(* Logix 5000 project; controller cal1615 1756-L62 rev 16.20; software revision 16.05; part 47 of 78 *)
(* tags used below, declared in another part *)
   FAULT : BOOL;   // Fault AFI
   HMI : BOOL;   // AFI HMI
   p01r03_lc3_ave_ctrl : CONTROL;
   p01r09_pb_global_reset : BOOL;   // System Modes PB: Global Fault Reset
   p02_real_from_hmi : hmi_real;   // MOP HMI Iface Real from HMI
   p22_ai_amps : REAL;   // Tension Stand 1 Analog Input Tension Stand 1 Motor Current
   p22_ai_hz : REAL;   // Tension Stand 1 Analog Input Tension Stand 1 Motor Hertz
   p22_ai_speed : REAL;
   p22_ai_ts1_lc : REAL;   // Tension Stand 1 Analog Input Loadcell
   p22_ao_selected_speed : REAL;   // Tension Stand 1 VFD Selected Speed
   p22_dint_to_hmi : DINT[16];   // Tension Stand 1 Dint to HMI
   p22_real_to_hmi : REAL[112];   // Tension Stand 1 Real to HMI
   p22r01 : routine;   // Tension Stand 1 Main
   p22r06 : routine;   // Tension Stand 1 Real to HMI
   p22r06_ave_lc : REAL;
   p22r06_lc_buffer : REAL[20];
   p22r06_lc_ctrl : CONTROL;
   p22r06_sample_timer : TIMER;
   p22r06_timer_fault : TIMER[4];   // Tension Stand 1 Real to HMI Fault Delay
   p22r06_timer_warning : TIMER[4];   // Tension Stand 1 Real to HMI Warning Delay
   p22r06_unload : DINT;
   p22r07 : routine;   // Tension Stand 1 Alarms
   p22r07_timer_fault : TIMER[4];   // Tension Stand 1 Alarms Fault Delay
   p22r07_timer_warning : TIMER[4];   // Tension Stand 1 Alarms Warning Delay
   p22r08 : routine;   // Tension Stand 1 Warnings
   p22r08_timer_fault : TIMER[4];   // Tension Stand 1 Warnings Fault Delay
   p22r08_timer_warning : TIMER[4];   // Tension Stand 1 Warnings Warning Delay
   p22r09 : routine;   // Tension Stand 1 Modes
   p22r11 : routine;   // Tension Stand 1 VFD
(* P22_Tension_Stand_1, continued *)

ROUTINE R06_Real_to_HMI   (* ladder *)
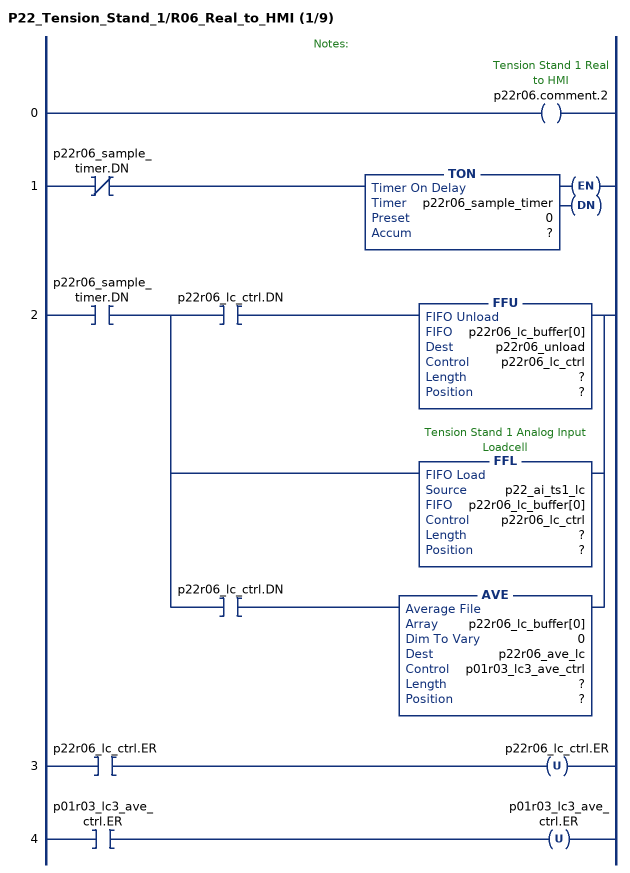
   // Notes:
   0: OTE(p22r06.comment.2);
   1: XIO(p22r06_sample_timer.DN)TON(p22r06_sample_timer,?,?);
   2: XIC(p22r06_sample_timer.DN)[XIC(p22r06_lc_ctrl.DN) FFU(p22r06_lc_buffer[0],p22r06_unload,p22r06_lc_ctrl,?,?) ,FFL(p22_ai_ts1_lc,p22r06_lc_buffer[0],p22r06_lc_ctrl,?,?) ,XIC(p22r06_lc_ctrl.DN) AVE(p22r06_lc_buffer[0],0,p22r06_ave_lc,p01r03_lc3_ave_ctrl,?,?) ];
   3: XIC(p22r06_lc_ctrl.ER)OTU(p22r06_lc_ctrl.ER);
   4: XIC(p01r03_lc3_ave_ctrl.ER)OTU(p01r03_lc3_ave_ctrl.ER);
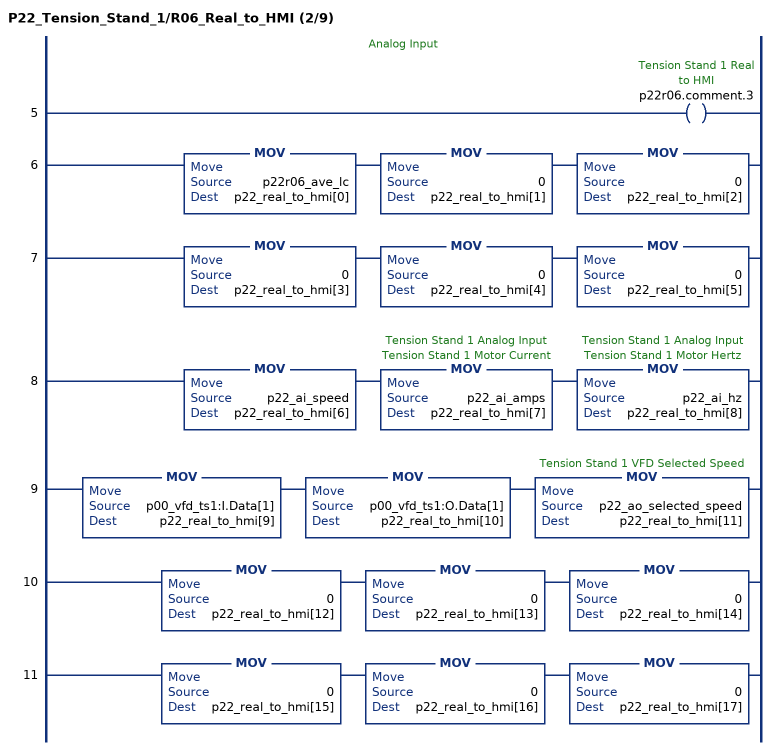
   // Analog Input
   5: OTE(p22r06.comment.3);
   6: MOV(p22r06_ave_lc,p22_real_to_hmi[0])MOV(0,p22_real_to_hmi[1])MOV(0,p22_real_to_hmi[2]);
   7: MOV(0,p22_real_to_hmi[3])MOV(0,p22_real_to_hmi[4])MOV(0,p22_real_to_hmi[5]);
   8: MOV(p22_ai_speed,p22_real_to_hmi[6])MOV(p22_ai_amps,p22_real_to_hmi[7])MOV(p22_ai_hz,p22_real_to_hmi[8]);
   9: MOV(p00_vfd_ts1:I.Data[1],p22_real_to_hmi[9])MOV(p00_vfd_ts1:O.Data[1],p22_real_to_hmi[10])MOV(p22_ao_selected_speed,p22_real_to_hmi[11]);
   10: MOV(0,p22_real_to_hmi[12])MOV(0,p22_real_to_hmi[13])MOV(0,p22_real_to_hmi[14]);
   11: MOV(0,p22_real_to_hmi[15])MOV(0,p22_real_to_hmi[16])MOV(0,p22_real_to_hmi[17]);
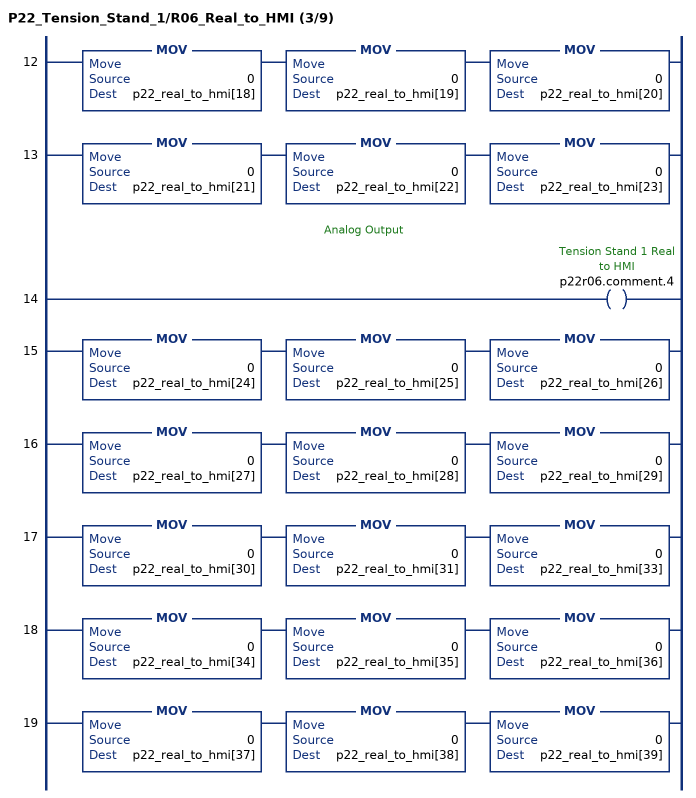
   12: MOV(0,p22_real_to_hmi[18])MOV(0,p22_real_to_hmi[19])MOV(0,p22_real_to_hmi[20]);
   13: MOV(0,p22_real_to_hmi[21])MOV(0,p22_real_to_hmi[22])MOV(0,p22_real_to_hmi[23]);
   // Analog Output
   14: OTE(p22r06.comment.4);
   15: MOV(0,p22_real_to_hmi[24])MOV(0,p22_real_to_hmi[25])MOV(0,p22_real_to_hmi[26]);
   16: MOV(0,p22_real_to_hmi[27])MOV(0,p22_real_to_hmi[28])MOV(0,p22_real_to_hmi[29]);
   17: MOV(0,p22_real_to_hmi[30])MOV(0,p22_real_to_hmi[31])MOV(0,p22_real_to_hmi[33]);
   18: MOV(0,p22_real_to_hmi[34])MOV(0,p22_real_to_hmi[35])MOV(0,p22_real_to_hmi[36]);
   19: MOV(0,p22_real_to_hmi[37])MOV(0,p22_real_to_hmi[38])MOV(0,p22_real_to_hmi[39]);
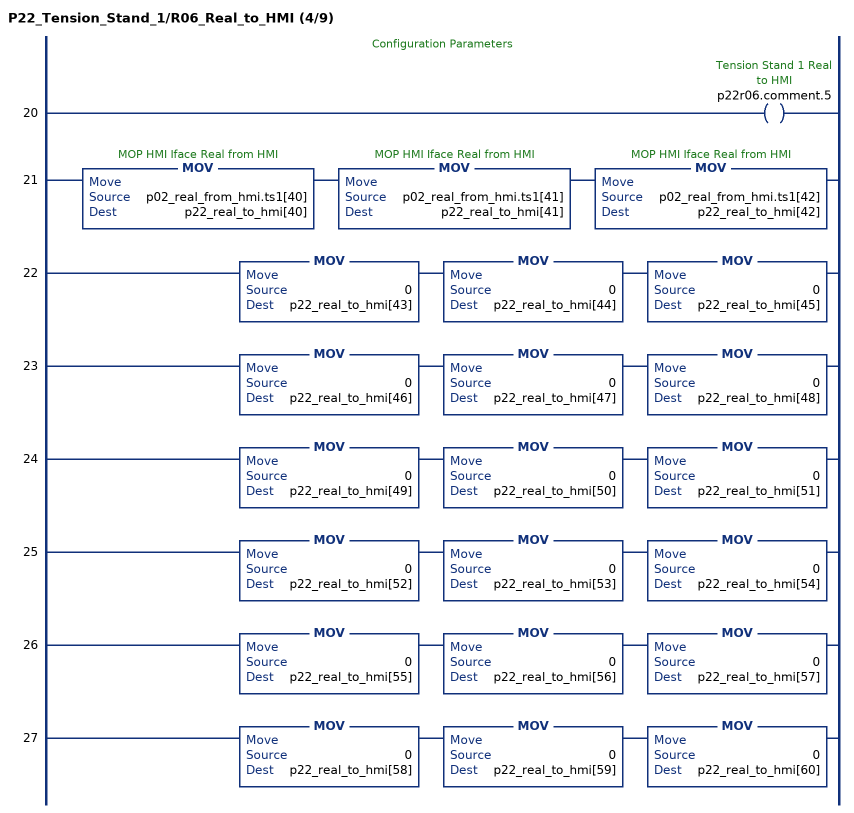
   // Configuration Parameters
   20: OTE(p22r06.comment.5);
   21: MOV(p02_real_from_hmi.ts1[40],p22_real_to_hmi[40])MOV(p02_real_from_hmi.ts1[41],p22_real_to_hmi[41])MOV(p02_real_from_hmi.ts1[42],p22_real_to_hmi[42]);
   22: MOV(0,p22_real_to_hmi[43])MOV(0,p22_real_to_hmi[44])MOV(0,p22_real_to_hmi[45]);
   23: MOV(0,p22_real_to_hmi[46])MOV(0,p22_real_to_hmi[47])MOV(0,p22_real_to_hmi[48]);
   24: MOV(0,p22_real_to_hmi[49])MOV(0,p22_real_to_hmi[50])MOV(0,p22_real_to_hmi[51]);
   25: MOV(0,p22_real_to_hmi[52])MOV(0,p22_real_to_hmi[53])MOV(0,p22_real_to_hmi[54]);
   26: MOV(0,p22_real_to_hmi[55])MOV(0,p22_real_to_hmi[56])MOV(0,p22_real_to_hmi[57]);
   27: MOV(0,p22_real_to_hmi[58])MOV(0,p22_real_to_hmi[59])MOV(0,p22_real_to_hmi[60]);
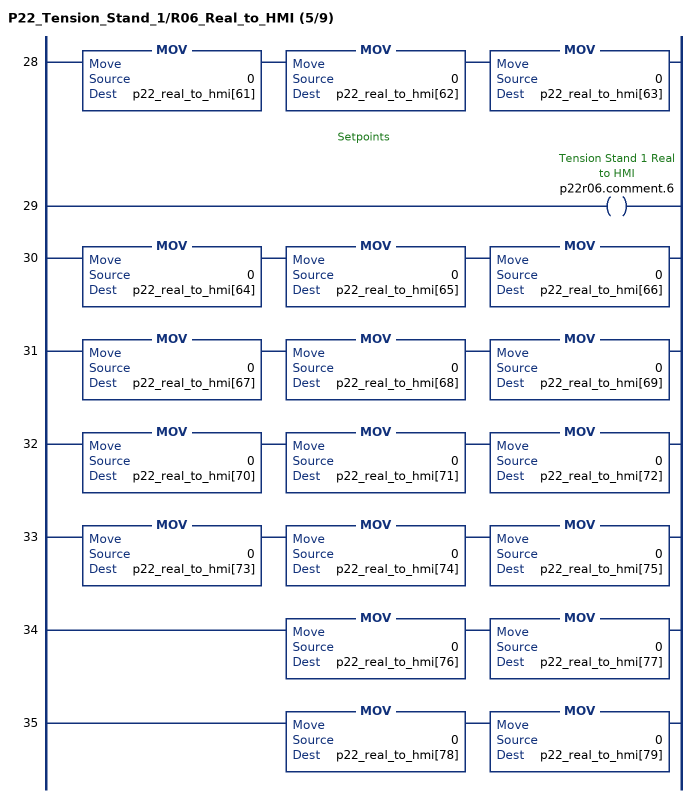
   28: MOV(0,p22_real_to_hmi[61])MOV(0,p22_real_to_hmi[62])MOV(0,p22_real_to_hmi[63]);
   // Setpoints
   29: OTE(p22r06.comment.6);
   30: MOV(0,p22_real_to_hmi[64])MOV(0,p22_real_to_hmi[65])MOV(0,p22_real_to_hmi[66]);
   31: MOV(0,p22_real_to_hmi[67])MOV(0,p22_real_to_hmi[68])MOV(0,p22_real_to_hmi[69]);
   32: MOV(0,p22_real_to_hmi[70])MOV(0,p22_real_to_hmi[71])MOV(0,p22_real_to_hmi[72]);
   33: MOV(0,p22_real_to_hmi[73])MOV(0,p22_real_to_hmi[74])MOV(0,p22_real_to_hmi[75]);
   34: MOV(0,p22_real_to_hmi[76])MOV(0,p22_real_to_hmi[77]);
   35: MOV(0,p22_real_to_hmi[78])MOV(0,p22_real_to_hmi[79]);
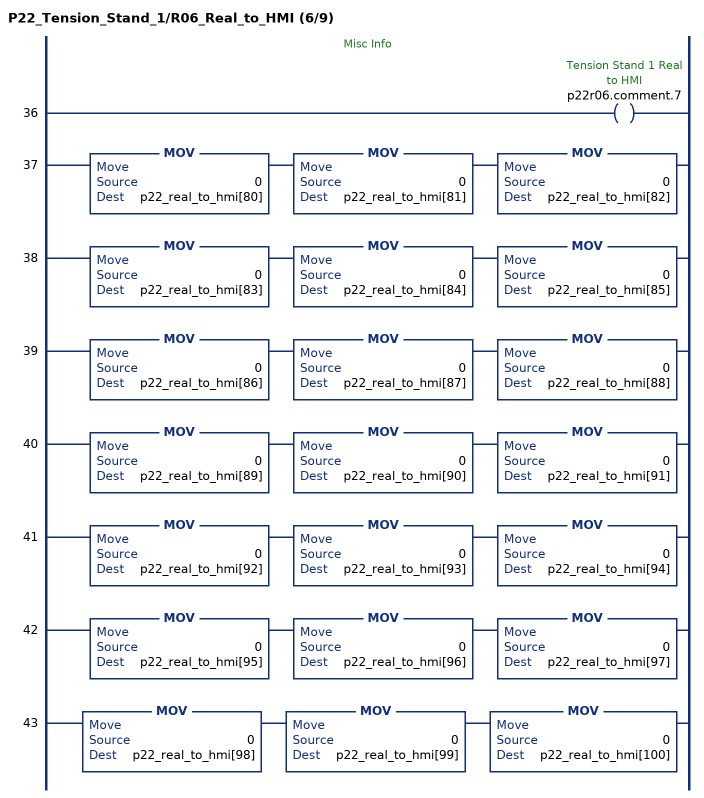
   // Misc Info
   36: OTE(p22r06.comment.7);
   37: MOV(0,p22_real_to_hmi[80])MOV(0,p22_real_to_hmi[81])MOV(0,p22_real_to_hmi[82]);
   38: MOV(0,p22_real_to_hmi[83])MOV(0,p22_real_to_hmi[84])MOV(0,p22_real_to_hmi[85]);
   39: MOV(0,p22_real_to_hmi[86])MOV(0,p22_real_to_hmi[87])MOV(0,p22_real_to_hmi[88]);
   40: MOV(0,p22_real_to_hmi[89])MOV(0,p22_real_to_hmi[90])MOV(0,p22_real_to_hmi[91]);
   41: MOV(0,p22_real_to_hmi[92])MOV(0,p22_real_to_hmi[93])MOV(0,p22_real_to_hmi[94]);
   42: MOV(0,p22_real_to_hmi[95])MOV(0,p22_real_to_hmi[96])MOV(0,p22_real_to_hmi[97]);
   43: MOV(0,p22_real_to_hmi[98])MOV(0,p22_real_to_hmi[99])MOV(0,p22_real_to_hmi[100]);
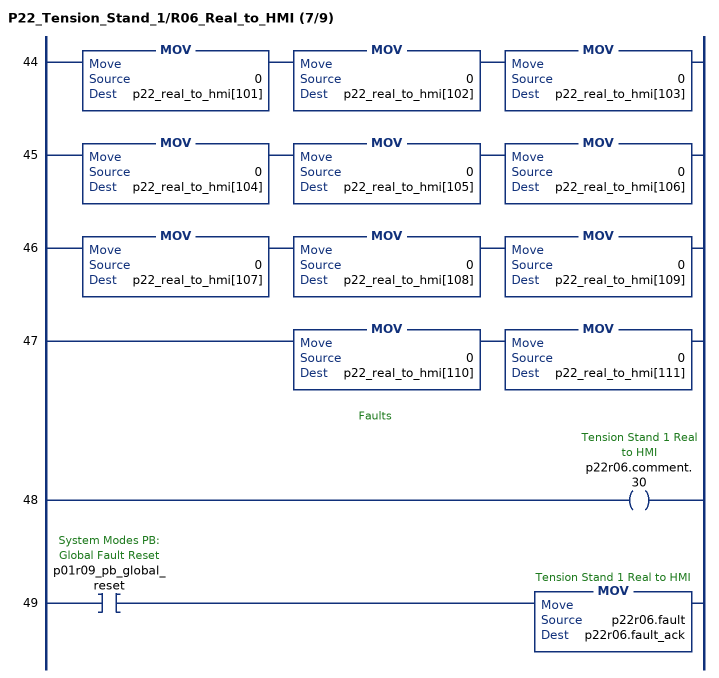
   44: MOV(0,p22_real_to_hmi[101])MOV(0,p22_real_to_hmi[102])MOV(0,p22_real_to_hmi[103]);
   45: MOV(0,p22_real_to_hmi[104])MOV(0,p22_real_to_hmi[105])MOV(0,p22_real_to_hmi[106]);
   46: MOV(0,p22_real_to_hmi[107])MOV(0,p22_real_to_hmi[108])MOV(0,p22_real_to_hmi[109]);
   47: MOV(0,p22_real_to_hmi[110])MOV(0,p22_real_to_hmi[111]);
   // Faults
   48: OTE(p22r06.comment.30);
   49: XIC(p01r09_pb_global_reset)MOV(p22r06.fault,p22r06.fault_ack);
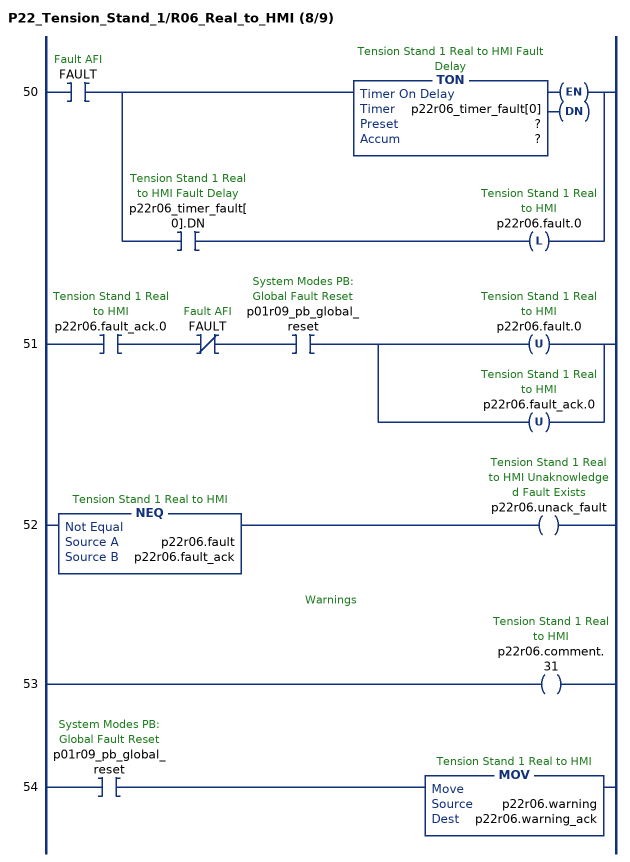
   50: XIC(FAULT)[TON(p22r06_timer_fault[0],?,?) ,XIC(p22r06_timer_fault[0].DN) OTL(p22r06.fault.0) ];
   51: XIC(p22r06.fault_ack.0)XIO(FAULT)XIC(p01r09_pb_global_reset)[OTU(p22r06.fault.0) ,OTU(p22r06.fault_ack.0) ];
   52: NEQ(p22r06.fault,p22r06.fault_ack)OTE(p22r06.unack_fault);
   // Warnings
   53: OTE(p22r06.comment.31);
   54: XIC(p01r09_pb_global_reset)MOV(p22r06.warning,p22r06.warning_ack);
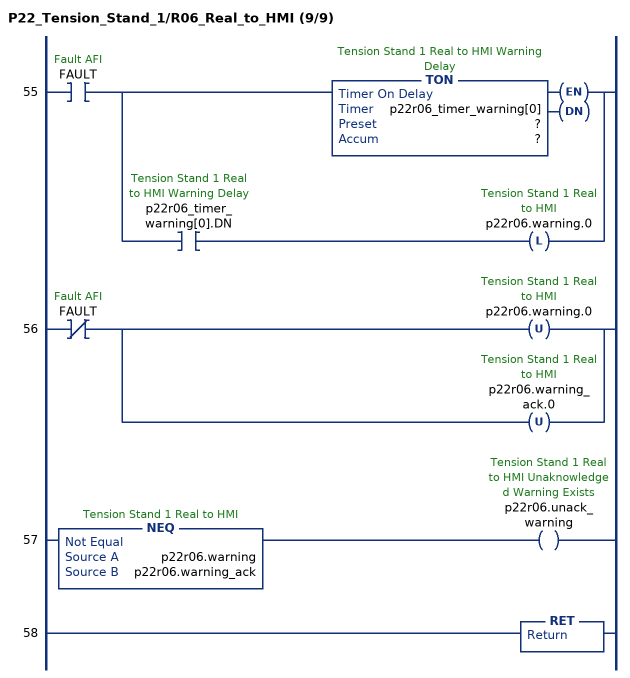
   55: XIC(FAULT)[TON(p22r06_timer_warning[0],?,?) ,XIC(p22r06_timer_warning[0].DN) OTL(p22r06.warning.0) ];
   56: XIO(FAULT)[OTU(p22r06.warning.0) ,OTU(p22r06.warning_ack.0) ];
   57: NEQ(p22r06.warning,p22r06.warning_ack)OTE(p22r06.unack_warning);
   58: RET();
END_ROUTINE

ROUTINE R07_Alarms   (* ladder *)
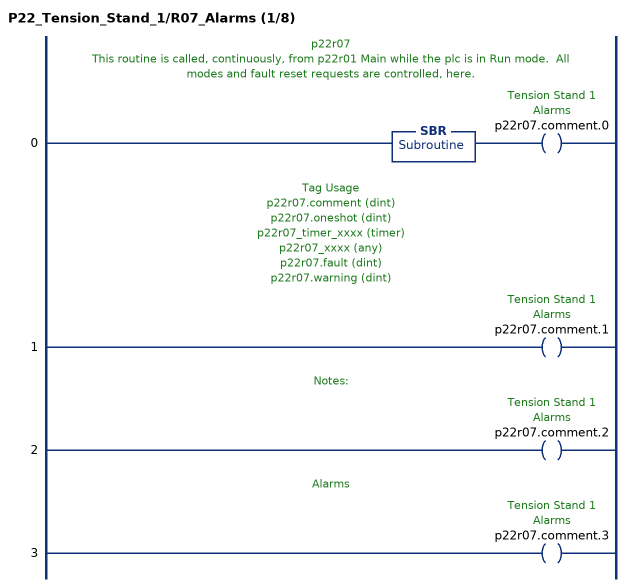
   // p22r07
   // This routine is called, continuously, from p22r01 Main while the plc is in Run mode.  All modes and fault reset requests are controlled, here.
   0: SBR()OTE(p22r07.comment.0);
   // Tag Usage
   // p22r07.comment (dint)
   // p22r07.oneshot (dint)
   // p22r07_timer_xxxx (timer)
   // p22r07_xxxx (any)
   // p22r07.fault (dint)
   // p22r07.warning (dint)
   1: OTE(p22r07.comment.1);
   // Notes:
   2: OTE(p22r07.comment.2);
   // Alarms
   3: OTE(p22r07.comment.3);
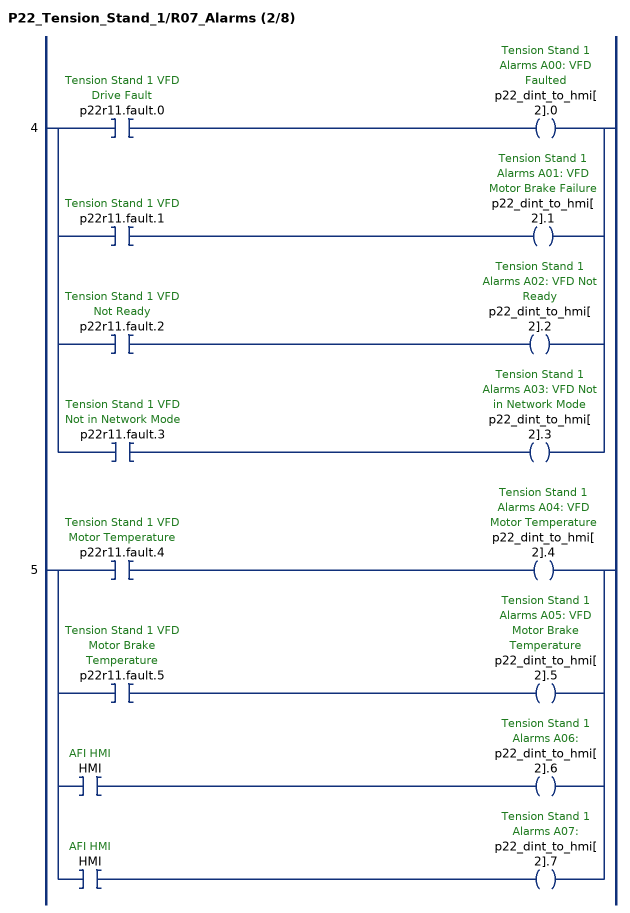
   4: [XIC(p22r11.fault.0) OTE(p22_dint_to_hmi[2].0) ,XIC(p22r11.fault.1) OTE(p22_dint_to_hmi[2].1) ,XIC(p22r11.fault.2) OTE(p22_dint_to_hmi[2].2) ,XIC(p22r11.fault.3) OTE(p22_dint_to_hmi[2].3) ];
   5: [XIC(p22r11.fault.4) OTE(p22_dint_to_hmi[2].4) ,XIC(p22r11.fault.5) OTE(p22_dint_to_hmi[2].5) ,XIC(HMI) OTE(p22_dint_to_hmi[2].6) ,XIC(HMI) OTE(p22_dint_to_hmi[2].7) ];
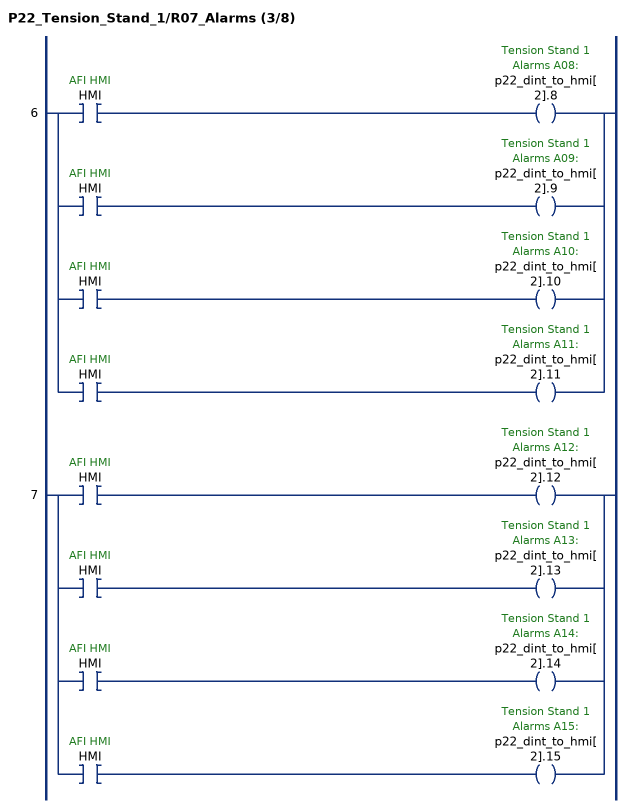
   6: [XIC(HMI) OTE(p22_dint_to_hmi[2].8) ,XIC(HMI) OTE(p22_dint_to_hmi[2].9) ,XIC(HMI) OTE(p22_dint_to_hmi[2].10) ,XIC(HMI) OTE(p22_dint_to_hmi[2].11) ];
   7: [XIC(HMI) OTE(p22_dint_to_hmi[2].12) ,XIC(HMI) OTE(p22_dint_to_hmi[2].13) ,XIC(HMI) OTE(p22_dint_to_hmi[2].14) ,XIC(HMI) OTE(p22_dint_to_hmi[2].15) ];
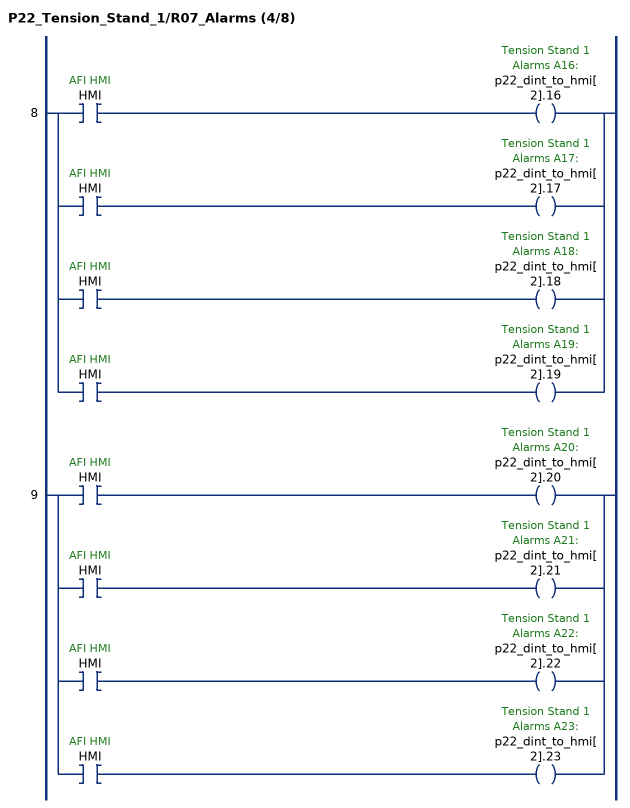
   8: [XIC(HMI) OTE(p22_dint_to_hmi[2].16) ,XIC(HMI) OTE(p22_dint_to_hmi[2].17) ,XIC(HMI) OTE(p22_dint_to_hmi[2].18) ,XIC(HMI) OTE(p22_dint_to_hmi[2].19) ];
   9: [XIC(HMI) OTE(p22_dint_to_hmi[2].20) ,XIC(HMI) OTE(p22_dint_to_hmi[2].21) ,XIC(HMI) OTE(p22_dint_to_hmi[2].22) ,XIC(HMI) OTE(p22_dint_to_hmi[2].23) ];
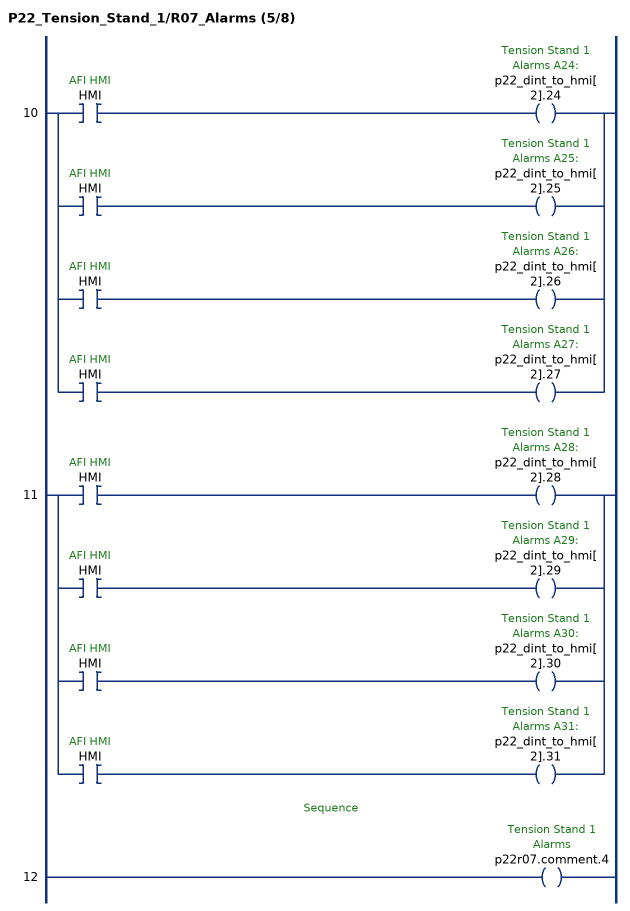
   10: [XIC(HMI) OTE(p22_dint_to_hmi[2].24) ,XIC(HMI) OTE(p22_dint_to_hmi[2].25) ,XIC(HMI) OTE(p22_dint_to_hmi[2].26) ,XIC(HMI) OTE(p22_dint_to_hmi[2].27) ];
   11: [XIC(HMI) OTE(p22_dint_to_hmi[2].28) ,XIC(HMI) OTE(p22_dint_to_hmi[2].29) ,XIC(HMI) OTE(p22_dint_to_hmi[2].30) ,XIC(HMI) OTE(p22_dint_to_hmi[2].31) ];
   // Sequence
   12: OTE(p22r07.comment.4);
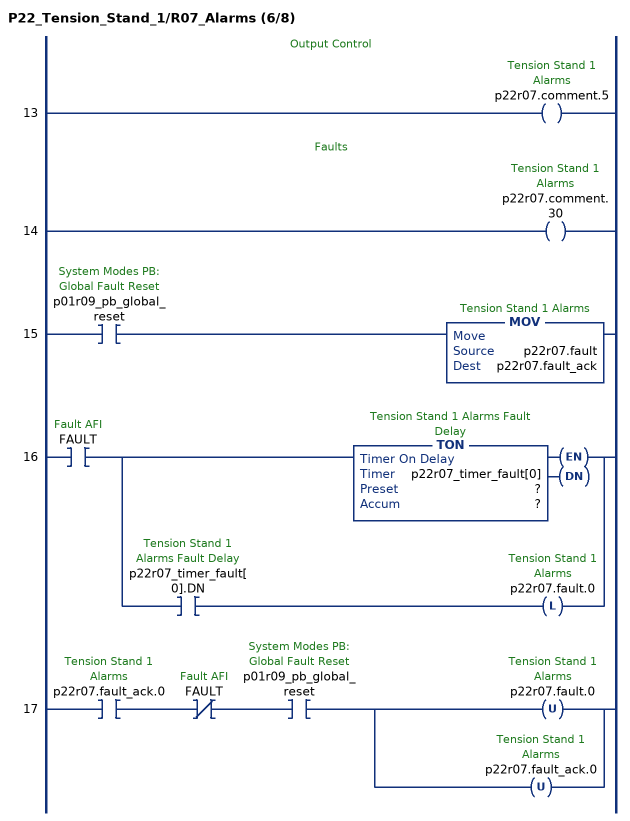
   // Output Control
   13: OTE(p22r07.comment.5);
   // Faults
   14: OTE(p22r07.comment.30);
   15: XIC(p01r09_pb_global_reset)MOV(p22r07.fault,p22r07.fault_ack);
   16: XIC(FAULT)[TON(p22r07_timer_fault[0],?,?) ,XIC(p22r07_timer_fault[0].DN) OTL(p22r07.fault.0) ];
   17: XIC(p22r07.fault_ack.0)XIO(FAULT)XIC(p01r09_pb_global_reset)[OTU(p22r07.fault.0) ,OTU(p22r07.fault_ack.0) ];
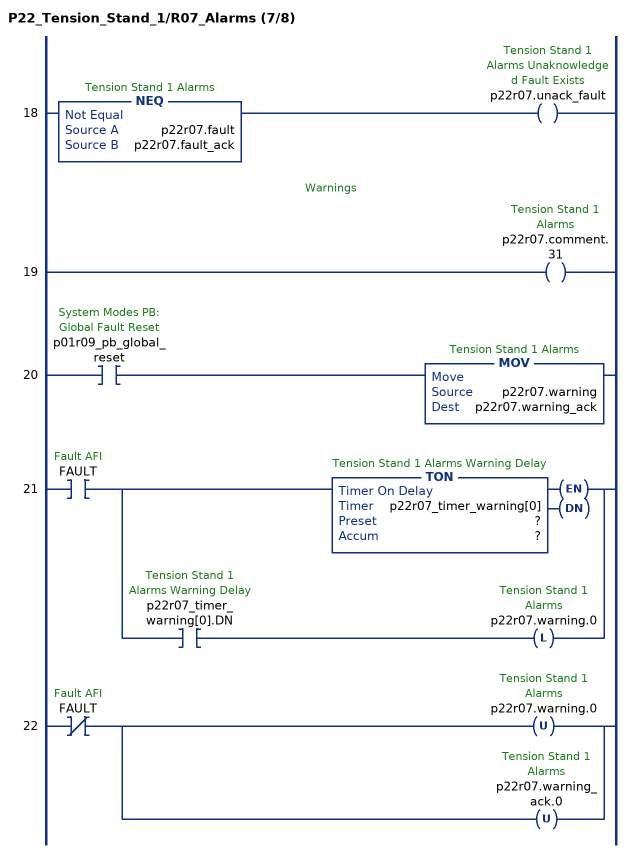
   18: NEQ(p22r07.fault,p22r07.fault_ack)OTE(p22r07.unack_fault);
   // Warnings
   19: OTE(p22r07.comment.31);
   20: XIC(p01r09_pb_global_reset)MOV(p22r07.warning,p22r07.warning_ack);
   21: XIC(FAULT)[TON(p22r07_timer_warning[0],?,?) ,XIC(p22r07_timer_warning[0].DN) OTL(p22r07.warning.0) ];
   22: XIO(FAULT)[OTU(p22r07.warning.0) ,OTU(p22r07.warning_ack.0) ];
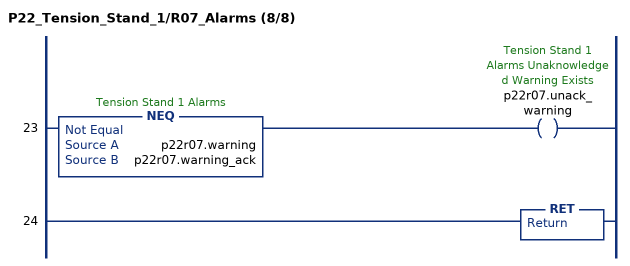
   23: NEQ(p22r07.warning,p22r07.warning_ack)OTE(p22r07.unack_warning);
   24: RET();
END_ROUTINE

ROUTINE R08_Warnings   (* ladder *)
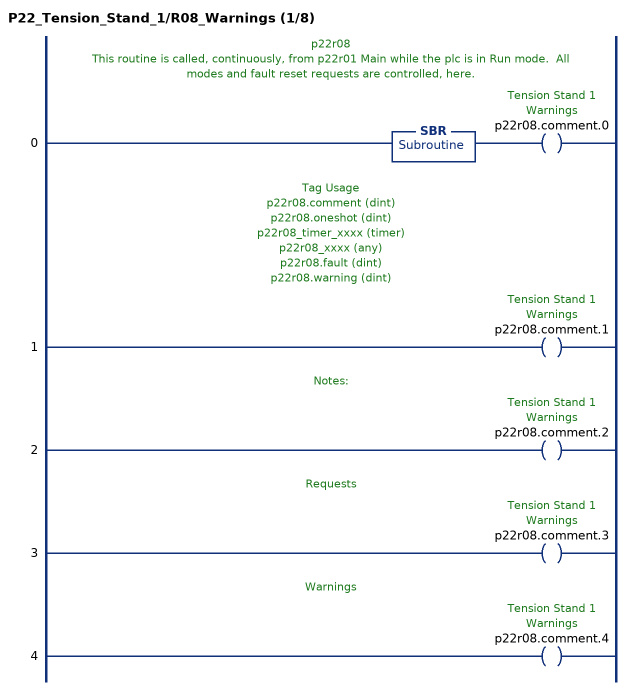
   // p22r08
   // This routine is called, continuously, from p22r01 Main while the plc is in Run mode.  All modes and fault reset requests are controlled, here.
   0: SBR()OTE(p22r08.comment.0);
   // Tag Usage
   // p22r08.comment (dint)
   // p22r08.oneshot (dint)
   // p22r08_timer_xxxx (timer)
   // p22r08_xxxx (any)
   // p22r08.fault (dint)
   // p22r08.warning (dint)
   1: OTE(p22r08.comment.1);
   // Notes:
   2: OTE(p22r08.comment.2);
   // Requests
   3: OTE(p22r08.comment.3);
   // Warnings
   4: OTE(p22r08.comment.4);
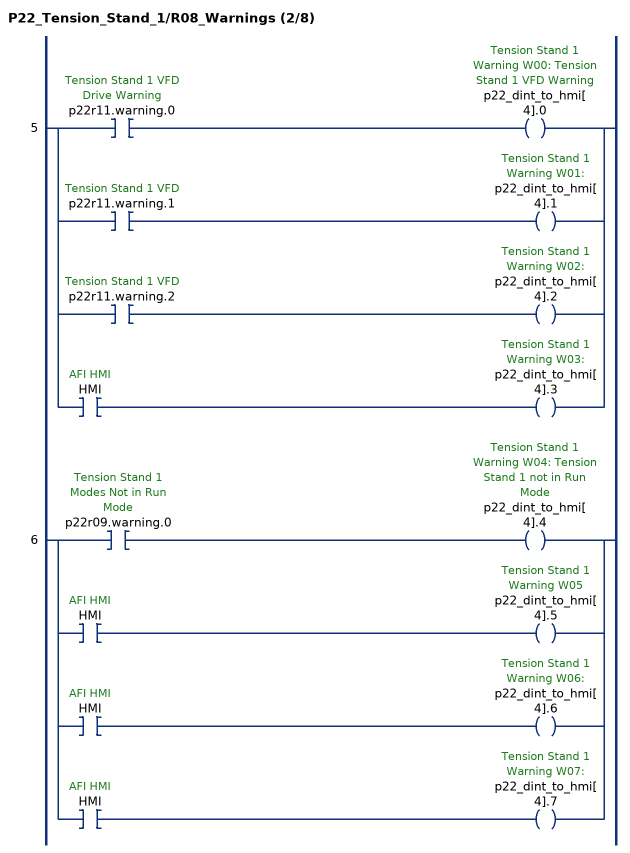
   5: [XIC(p22r11.warning.0) OTE(p22_dint_to_hmi[4].0) ,XIC(p22r11.warning.1) OTE(p22_dint_to_hmi[4].1) ,XIC(p22r11.warning.2) OTE(p22_dint_to_hmi[4].2) ,XIC(HMI) OTE(p22_dint_to_hmi[4].3) ];
   6: [XIC(p22r09.warning.0) OTE(p22_dint_to_hmi[4].4) ,XIC(HMI) OTE(p22_dint_to_hmi[4].5) ,XIC(HMI) OTE(p22_dint_to_hmi[4].6) ,XIC(HMI) OTE(p22_dint_to_hmi[4].7) ];
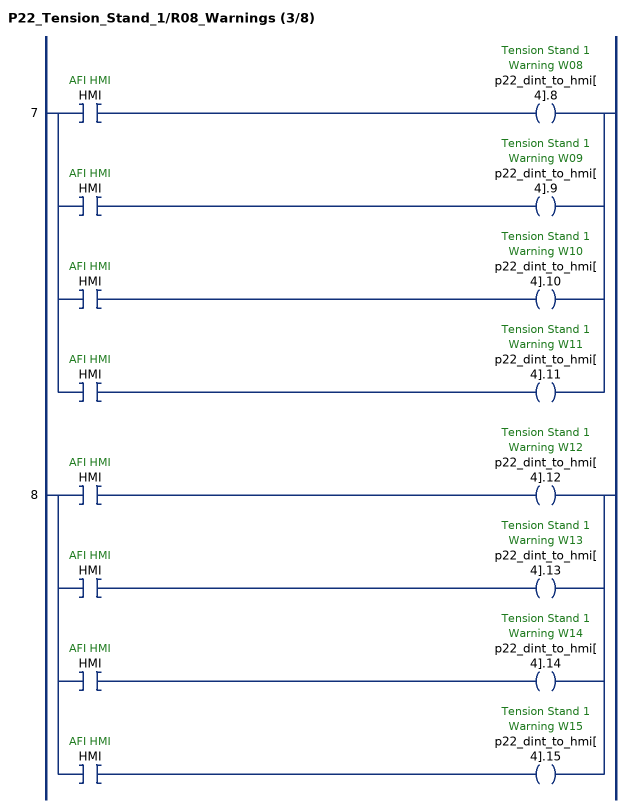
   7: [XIC(HMI) OTE(p22_dint_to_hmi[4].8) ,XIC(HMI) OTE(p22_dint_to_hmi[4].9) ,XIC(HMI) OTE(p22_dint_to_hmi[4].10) ,XIC(HMI) OTE(p22_dint_to_hmi[4].11) ];
   8: [XIC(HMI) OTE(p22_dint_to_hmi[4].12) ,XIC(HMI) OTE(p22_dint_to_hmi[4].13) ,XIC(HMI) OTE(p22_dint_to_hmi[4].14) ,XIC(HMI) OTE(p22_dint_to_hmi[4].15) ];
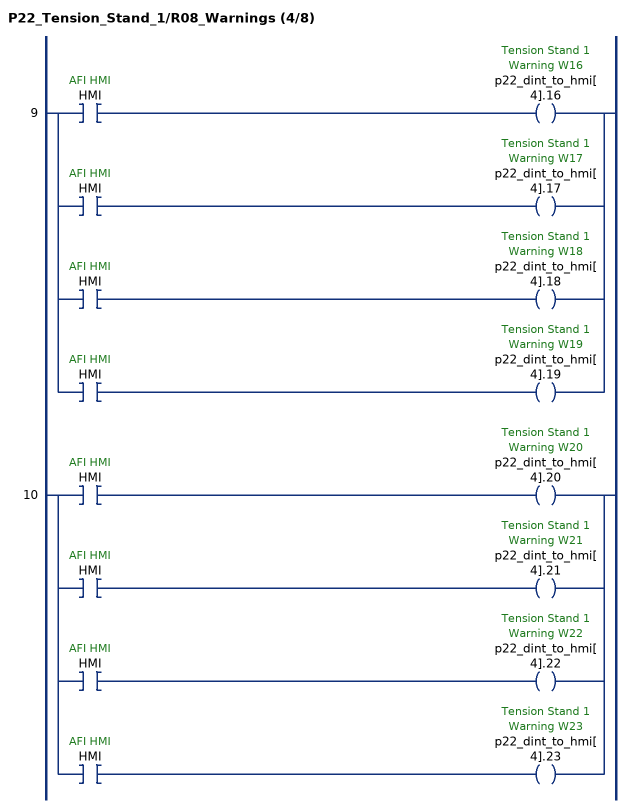
   9: [XIC(HMI) OTE(p22_dint_to_hmi[4].16) ,XIC(HMI) OTE(p22_dint_to_hmi[4].17) ,XIC(HMI) OTE(p22_dint_to_hmi[4].18) ,XIC(HMI) OTE(p22_dint_to_hmi[4].19) ];
   10: [XIC(HMI) OTE(p22_dint_to_hmi[4].20) ,XIC(HMI) OTE(p22_dint_to_hmi[4].21) ,XIC(HMI) OTE(p22_dint_to_hmi[4].22) ,XIC(HMI) OTE(p22_dint_to_hmi[4].23) ];
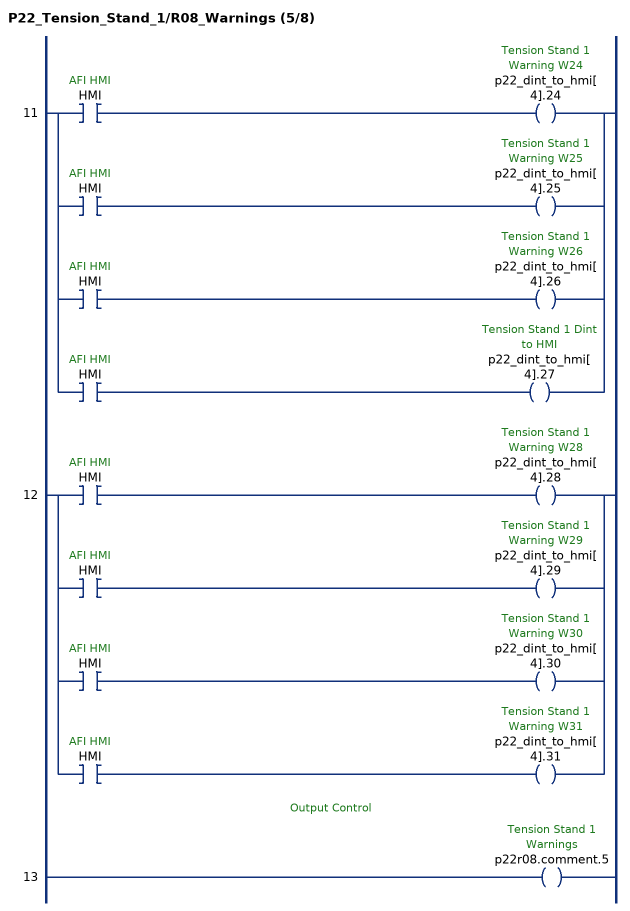
   11: [XIC(HMI) OTE(p22_dint_to_hmi[4].24) ,XIC(HMI) OTE(p22_dint_to_hmi[4].25) ,XIC(HMI) OTE(p22_dint_to_hmi[4].26) ,XIC(HMI) OTE(p22_dint_to_hmi[4].27) ];
   12: [XIC(HMI) OTE(p22_dint_to_hmi[4].28) ,XIC(HMI) OTE(p22_dint_to_hmi[4].29) ,XIC(HMI) OTE(p22_dint_to_hmi[4].30) ,XIC(HMI) OTE(p22_dint_to_hmi[4].31) ];
   // Output Control
   13: OTE(p22r08.comment.5);
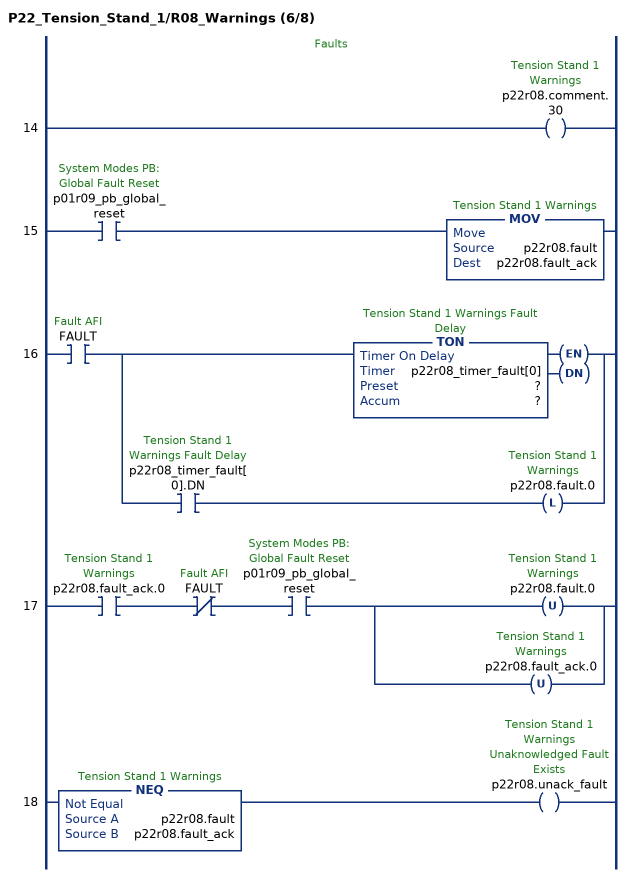
   // Faults
   14: OTE(p22r08.comment.30);
   15: XIC(p01r09_pb_global_reset)MOV(p22r08.fault,p22r08.fault_ack);
   16: XIC(FAULT)[TON(p22r08_timer_fault[0],?,?) ,XIC(p22r08_timer_fault[0].DN) OTL(p22r08.fault.0) ];
   17: XIC(p22r08.fault_ack.0)XIO(FAULT)XIC(p01r09_pb_global_reset)[OTU(p22r08.fault.0) ,OTU(p22r08.fault_ack.0) ];
   18: NEQ(p22r08.fault,p22r08.fault_ack)OTE(p22r08.unack_fault);
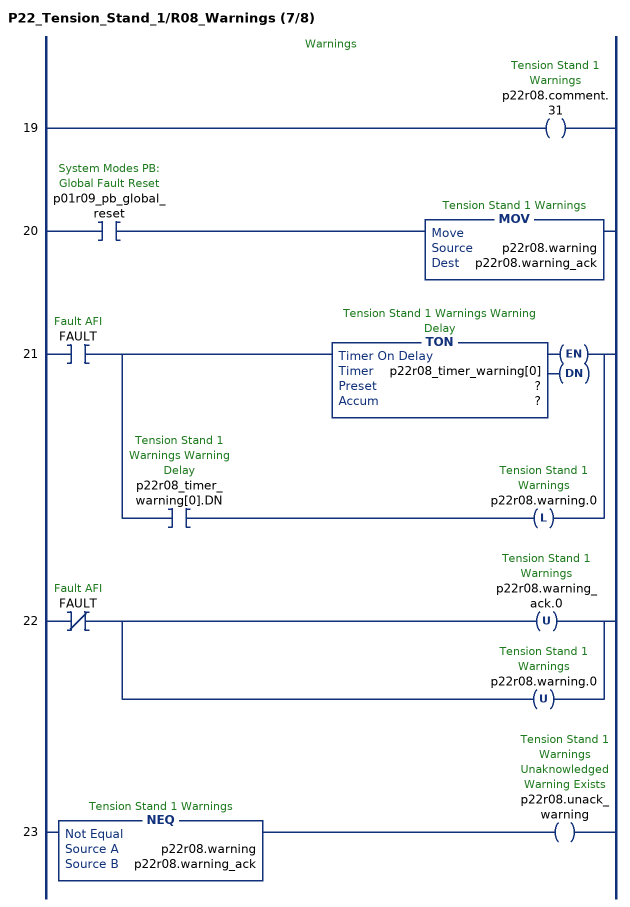
   // Warnings
   19: OTE(p22r08.comment.31);
   20: XIC(p01r09_pb_global_reset)MOV(p22r08.warning,p22r08.warning_ack);
   21: XIC(FAULT)[TON(p22r08_timer_warning[0],?,?) ,XIC(p22r08_timer_warning[0].DN) OTL(p22r08.warning.0) ];
   22: XIO(FAULT)[OTU(p22r08.warning_ack.0) ,OTU(p22r08.warning.0) ];
   23: NEQ(p22r08.warning,p22r08.warning_ack)OTE(p22r08.unack_warning);
